# EPICS autosave request: iocs/specsAnalyserIOC/iocBoot/iocSpecsAnalyser/auto_settings.req
file "ADBase_settings.req",       P=$(P),  R=cam1:
file "specsAnalyser.req",         P=$(P),  R=cam1:
file "NDStdArrays_settings.req",  P=$(P),  R=image1:
file "commonPlugin_settings.req", P=$(P)
